# B&R Automation Studio project ClaudeTest
Automation Studio 4.9

## Configuration Config1

CPU X20CP1686X, AutomationRuntime S4.93, Build 4.1.2, Vc V4.73.2

### Task classes (Cpu.sw)
```
Cyclic#4:
  TestPrg <- Source.TestPrg.prg
Libraries: standard
```

### Hardware
```
X20CP1686X : X20CP1686X v1.10.0.0
  Connector IF2:
    ActivateDevice = 1
  ConfigurationID = ClaudeTest_Config1
  Simulation = 1
  FileDevice1
  FileDeviceName1 = USER
  FileDevicePath1 = USER_PATH
```

## Logical view

### Global.var - Global variables
```iecst
VAR
	gSystemReady : BOOL;  (* przykładowa zmienna globalna *)
END_VAR

VAR CONSTANT

END_VAR
```

### Package Logical/Components - Custom project components (own FB libraries)

### Library Logical/Components/ActCtrl (IEC) - Actuator control function block.

#### ActCtrl.fun - Function block declaration
```iecst
FUNCTION_BLOCK ActCtrl
VAR_INPUT
	Cmd             : ActCtrlCmdType;
	Par             : ActCtrlParType;
	SensorRetracted : BOOL;  (* czujnik pozycji cofniętej *)
	SensorExtended  : BOOL;  (* czujnik pozycji wysuniętej *)
END_VAR
VAR_OUTPUT
	Sts : ActCtrlStsType;
END_VAR
VAR
	fbTimeout      : TON;
	ErrorLatch     : BOOL;
	SensorConflict : BOOL;
END_VAR
END_FUNCTION_BLOCK
```

#### ActCtrl.st - Function block implementation
```iecst
FUNCTION_BLOCK ActCtrl

SensorConflict := SensorRetracted AND SensorExtended;

Sts.Extended := SensorExtended AND NOT SensorRetracted;
Sts.Retracted := SensorRetracted AND NOT SensorExtended;
Sts.Moving := (Cmd.Extend AND NOT Sts.Extended) OR (NOT Cmd.Extend AND NOT Sts.Retracted);

fbTimeout(IN := Sts.Moving AND NOT ErrorLatch, PT := Par.MoveTimeout);

IF SensorConflict OR fbTimeout.Q THEN
	ErrorLatch := TRUE;
ELSIF Cmd.ErrorAcknowledge THEN
	ErrorLatch := FALSE;
END_IF;

Sts.Error := ErrorLatch;
Sts.Output := Cmd.Extend AND NOT Sts.Error;

END_FUNCTION_BLOCK
```

#### ActCtrl.typ - Library data types
```iecst
TYPE
	ActCtrlCmdType : STRUCT
		Extend           : BOOL;  (* TRUE = wysuń, FALSE = cofnij *)
		ErrorAcknowledge : BOOL;  (* kasowanie błędu *)
	END_STRUCT;
	ActCtrlParType : STRUCT
		MoveTimeout : TIME := T#5S;  (* maks. czas ruchu do pozycji docelowej *)
	END_STRUCT;
	ActCtrlStsType : STRUCT
		Output    : BOOL;  (* wyjście cyfrowe do siłownika: TRUE = wysuń, FALSE = cofnij *)
		Extended  : BOOL;  (* siłownik w pozycji wysuniętej *)
		Retracted : BOOL;  (* siłownik w pozycji cofniętej *)
		Moving    : BOOL;  (* siłownik w ruchu, pozycja docelowa jeszcze nie osiągnięta *)
		Error     : BOOL;  (* konflikt czujników lub przekroczony czas ruchu *)
	END_STRUCT;
END_TYPE
```

### Program Logical/Source/TestPrg (IEC)

#### Main.st - Init, cyclic, exit code
```iecst
PROGRAM _INIT
	(* Insert code here *)

END_PROGRAM

PROGRAM _CYCLIC
	(* symulacja czujników pozycji na podstawie wysterowania z ActCtrl - tylko do testów w ARsim *)
	fbActCtrlSim(Output := fbActCtrl.Sts.Output);

	fbActCtrl(
		SensorRetracted := fbActCtrlSim.SensorRetracted,
		SensorExtended  := fbActCtrlSim.SensorExtended
	);
END_PROGRAM

PROGRAM _EXIT
	(* Insert code here *)

END_PROGRAM
```

#### Variables.var - Local variables
```iecst
VAR
	fbActCtrl    : ActCtrl;
	fbActCtrlSim : ActCtrlSim;
END_VAR

VAR CONSTANT

END_VAR
```

#### ActCtrlSim.fun - Sensor simulation for ActCtrl (ARsim only) - declaration
```iecst
FUNCTION_BLOCK ActCtrlSim
VAR_INPUT
	Output     : BOOL;              (* wysterowanie z ActCtrl.Output: TRUE = wysuń, FALSE = cofnij *)
	TravelTime : TIME := T#2S;      (* symulowany czas przejazdu siłownika między pozycjami krańcowymi *)
END_VAR
VAR_OUTPUT
	SensorRetracted : BOOL;  (* symulowany Signal1 *)
	SensorExtended  : BOOL;  (* symulowany Signal2 *)
END_VAR
VAR
	fbExtendTravel  : TON;
	fbRetractTravel : TON;
END_VAR
END_FUNCTION_BLOCK
```

#### ActCtrlSim.st - Sensor simulation for ActCtrl (ARsim only) - implementation
```iecst
FUNCTION_BLOCK ActCtrlSim

fbExtendTravel(IN := Output, PT := TravelTime);
fbRetractTravel(IN := NOT Output, PT := TravelTime);

SensorExtended := fbExtendTravel.Q;
SensorRetracted := fbRetractTravel.Q;

END_FUNCTION_BLOCK
```

#### ActuatorControl.fun - not listed in the package file held
```iecst
FUNCTION_BLOCK FB_ActuatorControl
VAR_INPUT
	i_xCmdExtend    : BOOL;              (* TRUE = wysuń, FALSE = cofnij *)
	i_xSenRetracted : BOOL;              (* Signal1 - czujnik pozycji cofniętej *)
	i_xSenExtended  : BOOL;              (* Signal2 - czujnik pozycji wysuniętej *)
	i_xErrorAck     : BOOL;              (* kasowanie błędu *)
	i_tMoveTimeout  : TIME := T#5S;      (* maks. czas ruchu do pozycji docelowej *)
END_VAR
VAR_OUTPUT
	q_xOutput    : BOOL;  (* wyjście cyfrowe do siłownika: TRUE = wysuń, FALSE = cofnij *)
	q_xExtended  : BOOL;  (* siłownik w pozycji wysuniętej *)
	q_xRetracted : BOOL;  (* siłownik w pozycji cofniętej *)
	q_xMoving    : BOOL;  (* siłownik w ruchu, pozycja docelowa jeszcze nie osiągnięta *)
	q_xError     : BOOL;  (* konflikt czujników lub przekroczony czas ruchu *)
END_VAR
VAR
	fbTimeout      : TON;
	xErrorLatch    : BOOL;
	xSensorConflict: BOOL;
END_VAR
END_FUNCTION_BLOCK
```

#### ActuatorControl.st - not listed in the package file held
```iecst
FUNCTION_BLOCK FB_ActuatorControl

xSensorConflict := i_xSenRetracted AND i_xSenExtended;

q_xExtended  := i_xSenExtended AND NOT i_xSenRetracted;
q_xRetracted := i_xSenRetracted AND NOT i_xSenExtended;
q_xMoving    := (i_xCmdExtend AND NOT q_xExtended) OR (NOT i_xCmdExtend AND NOT q_xRetracted);

fbTimeout(IN := q_xMoving AND NOT xErrorLatch, PT := i_tMoveTimeout);

IF xSensorConflict OR fbTimeout.Q THEN
	xErrorLatch := TRUE;
ELSIF i_xErrorAck THEN
	xErrorLatch := FALSE;
END_IF;

q_xError  := xErrorLatch;
q_xOutput := i_xCmdExtend AND NOT q_xError;

END_FUNCTION_BLOCK
```

Listed in the project but not available here: Logical/Global.typ, Logical/Libraries, Logical/Components/ActCtrl/ActCtrl.var, Logical/Source/TestPrg/Types.typ
